// SIMATIC S7-200 project (STEP 7-Micro/WIN), CPU 224XP REL 02.01

SYMBOL_TABLE 用户定义1
                 AQW0     // 0-10V输出
END_SYMBOL_TABLE

ORGANIZATION_BLOCK 主程序:OB1
TITLE=【工贝电子】本测试程序适用于工贝电子兼容西门子PLC系列
// 
// 1.PLC的Port0口初始化为modbus rtu从站
// 2.Q点流水灯
// 3.每一秒钟VW10自加1
// 
BEGIN
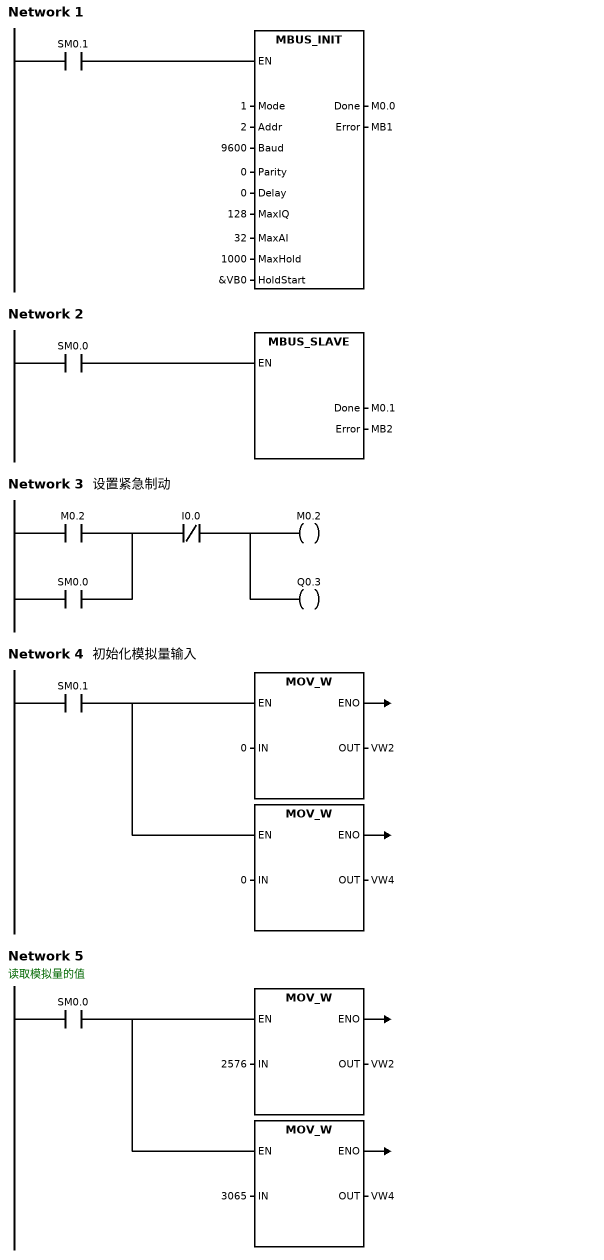
Network 1
LD     SM0.1
CALL   MBUS_INIT:SBR1, 1, 2, 9600, 0, 0, 128, 32, 1000, &VB0, M0.0, MB1
Network 2
LD     SM0.0
CALL   MBUS_SLAVE:SBR2, M0.1, MB2
Network 3 // 设置紧急制动
LD     M0.2
O      SM0.0
AN     I0.0
=      M0.2
=      Q0.3
Network 4 // 初始化模拟量输入
LD     SM0.1
MOVW   0, VW2
MOVW   0, VW4
Network 5
// 读取模拟量的值
LD     SM0.0
MOVW   2576, VW2
MOVW   3065, VW4
END_ORGANIZATION_BLOCK

// SBR1: protected block, not included

// SBR2: protected block, not included

// SBR3: protected block, not included

// SBR4: protected block, not included
